// TwinCAT 3 PLC project SPS_Program
// ProgramVersion: 3.1.4023.0
// libraries:
//   Tc2_EtherCAT, * (Beckhoff Automation GmbH)
//   Tc2_Standard, * (Beckhoff Automation GmbH)
//   Tc2_System, * (Beckhoff Automation GmbH)
//   Tc3_Module, * (Beckhoff Automation GmbH)
// project tree:
//   DUTs/ eStates.TcDUT
//   / PlcTask.TcTTO
//   POUs/ FB_EcMasterState.TcPOU, FB_IOs.TcPOU, FB_LightControl.TcPOU, FB_LogicSupply.TcPOU, FB_PowerSupply.TcPOU, FB_SlaveName.TcPOU, FB_Start.TcPOU, FB_WatchPhotoelectricBarrier.TcPOU, FB_YesNo.TcPOU, MAIN.TcPOU
// real-time tasks:
//   TASK PlcTask: cycle T#10ms, priority 20, ADS port 350
// I/O:
//   DEVICE Gerät 1 (Beckhoff CCAT)
//   DEVICE Gerät 2 (EtherCAT), AmsNetId 10.200.20.140.3.1
//     Klemme 1 (EK1200) [EK1200-5000 EtherCAT Netzteil (2A E-Bus)]
//       Klemme 2 (EL1018) [EL1018 8K. Dig. Eingang 24V, 10µs]
//       Klemme 3 (EL1018) [EL1018 8K. Dig. Eingang 24V, 10µs]
//       Klemme 4 (EL1018) [EL1018 8K. Dig. Eingang 24V, 10µs]
//       Klemme 5 (EL1018) [EL1018 8K. Dig. Eingang 24V, 10µs]
//       Klemme 6 (EL4104) [EL4104 4Ch. Ana. Ausgang 0-10V, 16bit]
//       Klemme 7 (EL3064) [EL3064 4Ch. Ana. Input 0-10V]
//       Klemme 8 (EL2068) [EL2068 8Ch. Dig Output 24V, 0.5A]
//       Klemme 9 (EL2068) [EL2068 8Ch. Dig Output 24V, 0.5A]
//       Klemme 10 (EL2068) [EL2068 8Ch. Dig Output 24V, 0.5A]
//       Klemme 11 (EL2068) [EL2068 8Ch. Dig Output 24V, 0.5A]
//       Klemme 12 (EL9011) [EL9011 Endklemme]
//   DEVICE Gerät 3 (EtherCAT), AmsNetId 10.200.20.140.4.1
//     Antrieb 14 (SOMANET Node) [SOMANET Node CiA402 Antrieb]
//       modules: Module 1 (CiA402 Dictionary)
//     Antrieb 15 (SOMANET Node) [SOMANET Node CiA402 Antrieb]
//       modules: Module 1 (CiA402 Dictionary)
// variable links:
//   SPS_Program/SPS_Program Instance <-> Device 2 (EtherCAT)/Term 1 (EK1200)/Term 10 (EL2068)
//     PlcTask Outputs/MAIN.bA83_1 <-> DOS RxPDO-Map Outputs Ch.01/Output
//     PlcTask Outputs/MAIN.bA83_2 <-> DOS RxPDO-Map Outputs Ch.03/Output
//     PlcTask Outputs/MAIN.bA83_3 <-> DOS RxPDO-Map Outputs Ch.05/Output
//     PlcTask Outputs/MAIN.bA83_4 <-> DOS RxPDO-Map Outputs Ch.07/Output
//     PlcTask Outputs/MAIN.bA83_5 <-> DOS RxPDO-Map Outputs Ch.02/Output
//     PlcTask Outputs/MAIN.bA83_6 <-> DOS RxPDO-Map Outputs Ch.04/Output
//     PlcTask Outputs/MAIN.bA83_7 <-> DOS RxPDO-Map Outputs Ch.06/Output
//     PlcTask Outputs/MAIN.bA83_8 <-> DOS RxPDO-Map Outputs Ch.08/Output
//   SPS_Program/SPS_Program Instance <-> Device 2 (EtherCAT)/Term 1 (EK1200)/Term 11 (EL2068)
//     PlcTask Outputs/MAIN.bA84_1 <-> DOS RxPDO-Map Outputs Ch.01/Output
//     PlcTask Outputs/MAIN.bA84_2 <-> DOS RxPDO-Map Outputs Ch.02/Output
//     PlcTask Outputs/MAIN.bA84_3 <-> DOS RxPDO-Map Outputs Ch.03/Output
//     PlcTask Outputs/MAIN.bA84_4 <-> DOS RxPDO-Map Outputs Ch.04/Output
//     PlcTask Outputs/MAIN.bA84_5 <-> DOS RxPDO-Map Outputs Ch.05/Output
//     PlcTask Outputs/MAIN.bA84_6 <-> DOS RxPDO-Map Outputs Ch.06/Output
//     PlcTask Outputs/MAIN.bA84_8 <-> DOS RxPDO-Map Outputs Ch.08/Output
//     PlcTask Outputs/MAIN.bA85_7 <-> DOS RxPDO-Map Outputs Ch.07/Output
//   SPS_Program/SPS_Program Instance <-> Device 2 (EtherCAT)/Term 1 (EK1200)/Term 2 (EL1018)
//     PlcTask Inputs/MAIN.bA61_1 <-> Channel 1/Input
//     PlcTask Inputs/MAIN.bA61_2 <-> Channel 3/Input
//     PlcTask Inputs/MAIN.bA61_3 <-> Channel 5/Input
//     PlcTask Inputs/MAIN.bA61_4 <-> Channel 7/Input
//     PlcTask Inputs/MAIN.bA61_5 <-> Channel 2/Input
//     PlcTask Inputs/MAIN.bA61_6 <-> Channel 4/Input
//     PlcTask Inputs/MAIN.bA61_7 <-> Channel 6/Input
//     PlcTask Inputs/MAIN.bA61_8 <-> Channel 8/Input
//   SPS_Program/SPS_Program Instance <-> Device 2 (EtherCAT)/Term 1 (EK1200)/Term 3 (EL1018)
//     PlcTask Inputs/MAIN.bA62_1 <-> Channel 1/Input
//   SPS_Program/SPS_Program Instance <-> Device 2 (EtherCAT)/Term 1 (EK1200)/Term 4 (EL1018)
//     PlcTask Inputs/MAIN.bA63_1 <-> Channel 1/Input
//   SPS_Program/SPS_Program Instance <-> Device 2 (EtherCAT)/Term 1 (EK1200)/Term 5 (EL1018)
//     PlcTask Inputs/MAIN.bA64_1 <-> Channel 1/Input
//     PlcTask Inputs/MAIN.bA64_2 <-> Channel 3/Input
//     PlcTask Inputs/MAIN.bA64_3 <-> Channel 5/Input
//     PlcTask Inputs/MAIN.bA64_4 <-> Channel 7/Input
//     PlcTask Inputs/MAIN.bA64_5 <-> Channel 2/Input
//     PlcTask Inputs/MAIN.bA64_6 <-> Channel 4/Input
//     PlcTask Inputs/MAIN.bA64_7 <-> Channel 6/Input
//     PlcTask Inputs/MAIN.bA64_8 <-> Channel 8/Input
//   SPS_Program/SPS_Program Instance <-> Device 2 (EtherCAT)/Term 1 (EK1200)/Term 6 (EL4104)
//     PlcTask Outputs/MAIN.nA71_1 <-> AO Output Channel 1/Analog output
//     PlcTask Outputs/MAIN.nA71_3 <-> AO Output Channel 3/Analog output
//     PlcTask Outputs/MAIN.nA71_5 <-> AO Output Channel 2/Analog output
//     PlcTask Outputs/MAIN.nA71_7 <-> AO Output Channel 4/Analog output
//   SPS_Program/SPS_Program Instance <-> Device 2 (EtherCAT)/Term 1 (EK1200)/Term 7 (EL3064)
//     PlcTask Inputs/MAIN.nA72_1 <-> AI Standard Channel 1/Value
//     PlcTask Inputs/MAIN.nA72_3 <-> AI Standard Channel 3/Value
//     PlcTask Inputs/MAIN.nA72_5 <-> AI Standard Channel 2/Value
//     PlcTask Inputs/MAIN.nA72_7 <-> AI Standard Channel 4/Value
//   SPS_Program/SPS_Program Instance <-> Device 2 (EtherCAT)/Term 1 (EK1200)/Term 8 (EL2068)
//     PlcTask Outputs/MAIN.bA81_1 <-> DOS RxPDO-Map Outputs Ch.01/Output
//     PlcTask Outputs/MAIN.bA81_2 <-> DOS RxPDO-Map Outputs Ch.03/Output
//     PlcTask Outputs/MAIN.bA81_3 <-> DOS RxPDO-Map Outputs Ch.05/Output
//     PlcTask Outputs/MAIN.bA81_4 <-> DOS RxPDO-Map Outputs Ch.07/Output
//     PlcTask Outputs/MAIN.bA81_5 <-> DOS RxPDO-Map Outputs Ch.02/Output
//     PlcTask Outputs/MAIN.bA81_6 <-> DOS RxPDO-Map Outputs Ch.04/Output
//     PlcTask Outputs/MAIN.bA81_7 <-> DOS RxPDO-Map Outputs Ch.06/Output
//     PlcTask Outputs/MAIN.bA81_8 <-> DOS RxPDO-Map Outputs Ch.08/Output
//   SPS_Program/SPS_Program Instance <-> Device 2 (EtherCAT)/Term 1 (EK1200)/Term 9 (EL2068)
//     PlcTask Outputs/MAIN.bA82_1 <-> DOS RxPDO-Map Outputs Ch.01/Output
//     PlcTask Outputs/MAIN.bA82_2 <-> DOS RxPDO-Map Outputs Ch.03/Output
//     PlcTask Outputs/MAIN.bA82_3 <-> DOS RxPDO-Map Outputs Ch.05/Output
//     PlcTask Outputs/MAIN.bA82_4 <-> DOS RxPDO-Map Outputs Ch.07/Output
//     PlcTask Outputs/MAIN.bA82_5 <-> DOS RxPDO-Map Outputs Ch.02/Output
//     PlcTask Outputs/MAIN.bA82_6 <-> DOS RxPDO-Map Outputs Ch.04/Output
//     PlcTask Outputs/MAIN.bA82_7 <-> DOS RxPDO-Map Outputs Ch.06/Output
//     PlcTask Outputs/MAIN.bA82_8 <-> DOS RxPDO-Map Outputs Ch.08/Output
//   SPS_Program/SPS_Program Instance <-> Device 3 (EtherCAT)/Drive 14 (SOMANET Node)
//     PlcTask Inputs/MAIN.statusword_node_13 <-> TxPDO Mapping 1/Statusword
//   SPS_Program/SPS_Program Instance <-> Device 3 (EtherCAT)/Drive 15 (SOMANET Node)
//     PlcTask Inputs/MAIN.statusword_node_14 <-> TxPDO Mapping 1/Statusword

CONFIGURATION SPS_Program
    RESOURCE PLC ON TwinCAT3
        TASK PlcTask(INTERVAL := T#10ms, PRIORITY := 20);
        PROGRAM MAIN WITH PlcTask : MAIN;
    END_RESOURCE
END_CONFIGURATION

// ---- DUTs/eStates.TcDUT
{attribute 'qualified_only'}
{attribute 'strict'}
TYPE eStates :
(
	INIT,
	START_EXECUTION,
	EXECUTING,
	DONE
);
END_TYPE

// ---- POUs/MAIN.TcPOU
PROGRAM MAIN
//A61
VAR
	{attribute 'TcLinkTo' := 'TIID^Device 2 (EtherCAT)^Term 1 (EK1200)^Term 2 (EL1018)^Channel 1^Input'} 
	bA61_1		AT %I* 				: BOOL;
	{attribute 'TcLinkTo' := 'TIID^Device 2 (EtherCAT)^Term 1 (EK1200)^Term 2 (EL1018)^Channel 3^Input'} 
	bA61_2		AT %I* 				: BOOL;
	{attribute 'TcLinkTo' := 'TIID^Device 2 (EtherCAT)^Term 1 (EK1200)^Term 2 (EL1018)^Channel 5^Input'} 
	bA61_3		AT %I* 				: BOOL; 
	{attribute 'TcLinkTo' := 'TIID^Device 2 (EtherCAT)^Term 1 (EK1200)^Term 2 (EL1018)^Channel 7^Input'} 	
	bA61_4		AT %I* 				: BOOL;	
	{attribute 'TcLinkTo' := 'TIID^Device 2 (EtherCAT)^Term 1 (EK1200)^Term 2 (EL1018)^Channel 2^Input'} 		
	bA61_5		AT %I* 				: BOOL;
	{attribute 'TcLinkTo' := 'TIID^Device 2 (EtherCAT)^Term 1 (EK1200)^Term 2 (EL1018)^Channel 4^Input'}	
	bA61_6		AT %I* 				: BOOL;
	{attribute 'TcLinkTo' := 'TIID^Device 2 (EtherCAT)^Term 1 (EK1200)^Term 2 (EL1018)^Channel 6^Input'}	
	bA61_7		AT %I* 				: BOOL;
	{attribute 'TcLinkTo' := 'TIID^Device 2 (EtherCAT)^Term 1 (EK1200)^Term 2 (EL1018)^Channel 8^Input'}
	bA61_8		AT %I* 				: BOOL;
	bSetEnable_SlaveName: BOOL;
END_VAR


//A62
VAR
	{attribute 'TcLinkTo' := 'TIID^Device 2 (EtherCAT)^Term 1 (EK1200)^Term 3 (EL1018)^Channel 1^Input'} 
	bA62_1		AT %I* 				: BOOL;
	{attribute 'TcLinkTo' := 'TIID^Device 3 (EtherCAT)^Term 1 (EK1200)^Term 3 (EL1018)^Channel 3^Input'} 
	bA62_2		AT %I* 				: BOOL;
	{attribute 'TcLinkTo' := 'TIID^Device 3 (EtherCAT)^Term 1 (EK1200)^Term 3 (EL1018)^Channel 5^Input'} 
	bA62_3		AT %I* 				: BOOL; 
	{attribute 'TcLinkTo' := 'TIID^Device 3 (EtherCAT)^Term 1 (EK1200)^Term 3 (EL1018)^Channel 7^Input'} 	
	bA62_4		AT %I* 				: BOOL;	
	{attribute 'TcLinkTo' := 'TIID^Device 3 (EtherCAT)^Term 1 (EK1200)^Term 3 (EL1018)^Channel 2^Input'} 		
	bA62_5		AT %I* 				: BOOL;
	{attribute 'TcLinkTo' := 'TIID^Device 3 (EtherCAT)^Term 1 (EK1200)^Term 3 (EL1018)^Channel 4^Input'}	
	bA62_6		AT %I* 				: BOOL;
	{attribute 'TcLinkTo' := 'TIID^Device 3 (EtherCAT)^Term 1 (EK1200)^Term 3 (EL1018)^Channel 6^Input'}	
	bA62_7		AT %I* 				: BOOL;
	{attribute 'TcLinkTo' := 'TIID^Device 3 (EtherCAT)^Term 1 (EK1200)^Term 3 (EL1018)^Channel 8^Input'}
	bA62_8		AT %I* 				: BOOL;
END_VAR


//A63
VAR
	{attribute 'TcLinkTo' := 'TIID^Device 2 (EtherCAT)^Term 1 (EK1200)^Term 4 (EL1018)^Channel 1^Input'} 
	bA63_1		AT %I* 				: BOOL;
	{attribute 'TcLinkTo' := 'TIID^Device 3 (EtherCAT)^Term 1 (EK1200)^Term 4 (EL1018)^Channel 3^Input'} 
	bA63_2		AT %I* 				: BOOL;
	{attribute 'TcLinkTo' := 'TIID^Device 3 (EtherCAT)^Term 1 (EK1200)^Term 4 (EL1018)^Channel 5^Input'} 
	bA63_3		AT %I* 				: BOOL; 
	{attribute 'TcLinkTo' := 'TIID^Device 3 (EtherCAT)^Term 1 (EK1200)^Term 4 (EL1018)^Channel 7^Input'} 	
	bA63_4		AT %I* 				: BOOL;	
	{attribute 'TcLinkTo' := 'TIID^Device 3 (EtherCAT)^Term 1 (EK1200)^Term 4 (EL1018)^Channel 2^Input'} 		
	bA63_5		AT %I* 				: BOOL;
	{attribute 'TcLinkTo' := 'TIID^Device 3 (EtherCAT)^Term 1 (EK1200)^Term 4 (EL1018)^Channel 4^Input'}	
	bA63_6		AT %I* 				: BOOL;
	{attribute 'TcLinkTo' := 'TIID^Device 3 (EtherCAT)^Term 1 (EK1200)^Term 4 (EL1018)^Channel 6^Input'}	
	bA63_7		AT %I* 				: BOOL;
	{attribute 'TcLinkTo' := 'TIID^Device 3 (EtherCAT)^Term 1 (EK1200)^Term 4 (EL1018)^Channel 8^Input'}
	bA63_8		AT %I* 				: BOOL;
END_VAR


//A64
VAR
	{attribute 'TcLinkTo' := 'TIID^Device 2 (EtherCAT)^Term 1 (EK1200)^Term 5 (EL1018)^Channel 1^Input'}
	bA64_1		AT %I*				: BOOL; 
	{attribute 'TcLinkTo' := 'TIID^Device 2 (EtherCAT)^Term 1 (EK1200)^Term 5 (EL1018)^Channel 3^Input'}	
	bA64_2		AT %I* 				: BOOL;	
	{attribute 'TcLinkTo' := 'TIID^Device 2 (EtherCAT)^Term 1 (EK1200)^Term 5 (EL1018)^Channel 5^Input'}
	bA64_3		AT %I* 				: BOOL;
	{attribute 'TcLinkTo' := 'TIID^Device 2 (EtherCAT)^Term 1 (EK1200)^Term 5 (EL1018)^Channel 7^Input'}
	bA64_4		AT %I* 				: BOOL;
	{attribute 'TcLinkTo' := 'TIID^Device 2 (EtherCAT)^Term 1 (EK1200)^Term 5 (EL1018)^Channel 2^Input'}
	bA64_5		AT %I* 				: BOOL;
	{attribute 'TcLinkTo' := 'TIID^Device 2 (EtherCAT)^Term 1 (EK1200)^Term 5 (EL1018)^Channel 4^Input'}
	bA64_6		AT %I* 				: BOOL;
	{attribute 'TcLinkTo' := 'TIID^Device 2 (EtherCAT)^Term 1 (EK1200)^Term 5 (EL1018)^Channel 6^Input'}	
	bA64_7		AT %I* 				: BOOL;
	{attribute 'TcLinkTo' := 'TIID^Device 2 (EtherCAT)^Term 1 (EK1200)^Term 5 (EL1018)^Channel 8^Input'}
	bA64_8		AT %I* 				: BOOL;	
END_VAR


//A71
VAR	
	{attribute 'TcLinkTo' := 'TIID^Device 2 (EtherCAT)^Term 1 (EK1200)^Term 6 (EL4104)^AO Output Channel 1^Analog output'} 
	nA71_1		AT %Q* 				: UINT;
	{attribute 'TcLinkTo' := 'TIID^Device 2 (EtherCAT)^Term 1 (EK1200)^Term 6 (EL4104)^AO Output Channel 3^Analog output'} 
	nA71_3		AT %Q* 				: UINT;	
	{attribute 'TcLinkTo' := 'TIID^Device 2 (EtherCAT)^Term 1 (EK1200)^Term 6 (EL4104)^AO Output Channel 2^Analog output'} 
	nA71_5		AT %Q* 				: UINT;	
	{attribute 'TcLinkTo' := 'TIID^Device 2 (EtherCAT)^Term 1 (EK1200)^Term 6 (EL4104)^AO Output Channel 4^Analog output'} 
	nA71_7		AT %Q* 				: UINT;		
END_VAR


//A72
VAR
	{attribute 'TcLinkTo' := 'TIID^Device 2 (EtherCAT)^Term 1 (EK1200)^Term 7 (EL3064)^AI Standard Channel 1^Value'}
	nA72_1		AT %I* 				: UINT;	
	{attribute 'TcLinkTo' := 'TIID^Device 2 (EtherCAT)^Term 1 (EK1200)^Term 7 (EL3064)^AI Standard Channel 3^Value'}
 	nA72_3		AT %I* 				: UINT;	
	{attribute 'TcLinkTo' := 'TIID^Device 2 (EtherCAT)^Term 1 (EK1200)^Term 7 (EL3064)^AI Standard Channel 2^Value'}
	nA72_5		AT %I* 				: UINT;
	{attribute 'TcLinkTo' := 'TIID^Device 2 (EtherCAT)^Term 1 (EK1200)^Term 7 (EL3064)^AI Standard Channel 4^Value'}	
	nA72_7		AT %I* 				: UINT;	
END_VAR


//A81
VAR
	{attribute 'TcLinkTo' := 'TIID^Device 2 (EtherCAT)^Term 1 (EK1200)^Term 8 (EL2068)^DOS RxPDO-Map Outputs Ch.01^Output'}	
	bA81_1		AT %Q* 				: BOOL;
	{attribute 'TcLinkTo' := 'TIID^Device 2 (EtherCAT)^Term 1 (EK1200)^Term 8 (EL2068)^DOS RxPDO-Map Outputs Ch.03^Output'}		
	bA81_2		AT %Q* 				: BOOL;
	{attribute 'TcLinkTo' := 'TIID^Device 2 (EtherCAT)^Term 1 (EK1200)^Term 8 (EL2068)^DOS RxPDO-Map Outputs Ch.05^Output'}		
	bA81_3		AT %Q* 				: BOOL;
	{attribute 'TcLinkTo' := 'TIID^Device 2 (EtherCAT)^Term 1 (EK1200)^Term 8 (EL2068)^DOS RxPDO-Map Outputs Ch.07^Output'} 
	bA81_4		AT %Q* 				: BOOL; 
	{attribute 'TcLinkTo' := 'TIID^Device 2 (EtherCAT)^Term 1 (EK1200)^Term 8 (EL2068)^DOS RxPDO-Map Outputs Ch.02^Output'}
	bA81_5		AT %Q* 				: BOOL; 
	{attribute 'TcLinkTo' := 'TIID^Device 2 (EtherCAT)^Term 1 (EK1200)^Term 8 (EL2068)^DOS RxPDO-Map Outputs Ch.04^Output'}
	bA81_6		AT %Q* 				: BOOL;	
	{attribute 'TcLinkTo' := 'TIID^Device 2 (EtherCAT)^Term 1 (EK1200)^Term 8 (EL2068)^DOS RxPDO-Map Outputs Ch.06^Output'}
	bA81_7		AT %Q* 				: BOOL; 
	{attribute 'TcLinkTo' := 'TIID^Device 2 (EtherCAT)^Term 1 (EK1200)^Term 8 (EL2068)^DOS RxPDO-Map Outputs Ch.08^Output'}
	bA81_8		AT %Q* 				: BOOL; 
END_VAR


//A82
VAR
	{attribute 'TcLinkTo' := 'TIID^Device 2 (EtherCAT)^Term 1 (EK1200)^Term 9 (EL2068)^DOS RxPDO-Map Outputs Ch.01^Output'}
	bA82_1		AT %Q* 				: BOOL;
	{attribute 'TcLinkTo' := 'TIID^Device 2 (EtherCAT)^Term 1 (EK1200)^Term 9 (EL2068)^DOS RxPDO-Map Outputs Ch.03^Output'}
	bA82_2		AT %Q* 				: BOOL;
	{attribute 'TcLinkTo' := 'TIID^Device 2 (EtherCAT)^Term 1 (EK1200)^Term 9 (EL2068)^DOS RxPDO-Map Outputs Ch.05^Output'}
	bA82_3		AT %Q* 				: BOOL;
	{attribute 'TcLinkTo' := 'TIID^Device 2 (EtherCAT)^Term 1 (EK1200)^Term 9 (EL2068)^DOS RxPDO-Map Outputs Ch.07^Output'}
	bA82_4		AT %Q* 				: BOOL;
	{attribute 'TcLinkTo' := 'TIID^Device 2 (EtherCAT)^Term 1 (EK1200)^Term 9 (EL2068)^DOS RxPDO-Map Outputs Ch.02^Output'}
	bA82_5		AT %Q* 				: BOOL;
	{attribute 'TcLinkTo' := 'TIID^Device 2 (EtherCAT)^Term 1 (EK1200)^Term 9 (EL2068)^DOS RxPDO-Map Outputs Ch.04^Output'}
	bA82_6		AT %Q* 				: BOOL;
	{attribute 'TcLinkTo' := 'TIID^Device 2 (EtherCAT)^Term 1 (EK1200)^Term 9 (EL2068)^DOS RxPDO-Map Outputs Ch.06^Output'}
	bA82_7		AT %Q* 				: BOOL;
	{attribute 'TcLinkTo' := 'TIID^Device 2 (EtherCAT)^Term 1 (EK1200)^Term 9 (EL2068)^DOS RxPDO-Map Outputs Ch.08^Output'}
	bA82_8		AT %Q* 				: BOOL;
END_VAR


//A83
VAR
	{attribute 'TcLinkTo' := 'TIID^Device 2 (EtherCAT)^Term 1 (EK1200)^Term 10 (EL2068)^DOS RxPDO-Map Outputs Ch.01^Output'}
	bA83_1		AT %Q* 				: BOOL;
	{attribute 'TcLinkTo' := 'TIID^Device 2 (EtherCAT)^Term 1 (EK1200)^Term 10 (EL2068)^DOS RxPDO-Map Outputs Ch.03^Output'}
	bA83_2		AT %Q* 				: BOOL;
	{attribute 'TcLinkTo' := 'TIID^Device 2 (EtherCAT)^Term 1 (EK1200)^Term 10 (EL2068)^DOS RxPDO-Map Outputs Ch.05^Output'}
	bA83_3		AT %Q* 				: BOOL;
	{attribute 'TcLinkTo' := 'TIID^Device 2 (EtherCAT)^Term 1 (EK1200)^Term 10 (EL2068)^DOS RxPDO-Map Outputs Ch.07^Output'}
	bA83_4		AT %Q* 				: BOOL;
	{attribute 'TcLinkTo' := 'TIID^Device 2 (EtherCAT)^Term 1 (EK1200)^Term 10 (EL2068)^DOS RxPDO-Map Outputs Ch.02^Output'}
	bA83_5		AT %Q* 				: BOOL;
	{attribute 'TcLinkTo' := 'TIID^Device 2 (EtherCAT)^Term 1 (EK1200)^Term 10 (EL2068)^DOS RxPDO-Map Outputs Ch.04^Output'}
	bA83_6		AT %Q* 				: BOOL;
	{attribute 'TcLinkTo' := 'TIID^Device 2 (EtherCAT)^Term 1 (EK1200)^Term 10 (EL2068)^DOS RxPDO-Map Outputs Ch.06^Output'}
	bA83_7		AT %Q* 				: BOOL;
	{attribute 'TcLinkTo' := 'TIID^Device 2 (EtherCAT)^Term 1 (EK1200)^Term 10 (EL2068)^DOS RxPDO-Map Outputs Ch.08^Output'}
	bA83_8		AT %Q* 				: BOOL;	
END_VAR


//A84
//TODO
VAR	
	{attribute 'TcLinkTo' := 'TIID^Device 2 (EtherCAT)^Term 1 (EK1200)^Term 11 (EL2068)^DOS RxPDO-Map Outputs Ch.01^Output'}
	bA84_1		AT %Q* 				: BOOL;
	{attribute 'TcLinkTo' := 'TIID^Device 2 (EtherCAT)^Term 1 (EK1200)^Term 11 (EL2068)^DOS RxPDO-Map Outputs Ch.02^Output'}
	bA84_2		AT %Q* 				: BOOL;
	{attribute 'TcLinkTo' := 'TIID^Device 2 (EtherCAT)^Term 1 (EK1200)^Term 11 (EL2068)^DOS RxPDO-Map Outputs Ch.03^Output'}
	bA84_3		AT %Q* 				: BOOL;	
	{attribute 'TcLinkTo' := 'TIID^Device 2 (EtherCAT)^Term 1 (EK1200)^Term 11 (EL2068)^DOS RxPDO-Map Outputs Ch.04^Output'}
	bA84_4		AT %Q* 				: BOOL;
	{attribute 'TcLinkTo' := 'TIID^Device 2 (EtherCAT)^Term 1 (EK1200)^Term 11 (EL2068)^DOS RxPDO-Map Outputs Ch.05^Output'}
	bA84_5		AT %Q* 				: BOOL;
	{attribute 'TcLinkTo' := 'TIID^Device 2 (EtherCAT)^Term 1 (EK1200)^Term 11 (EL2068)^DOS RxPDO-Map Outputs Ch.06^Output'}
	bA84_6		AT %Q* 				: BOOL;
	{attribute 'TcLinkTo' := 'TIID^Device 2 (EtherCAT)^Term 1 (EK1200)^Term 11 (EL2068)^DOS RxPDO-Map Outputs Ch.07^Output'}
	bA85_7		AT %Q* 				: BOOL;
	{attribute 'TcLinkTo' := 'TIID^Device 2 (EtherCAT)^Term 1 (EK1200)^Term 11 (EL2068)^DOS RxPDO-Map Outputs Ch.08^Output'}
	bA84_8		AT %Q* 				: BOOL;
END_VAR

VAR
	fbLightControlLeft				: FB_LightControl;
	fbLightControlRight				: FB_LightControl;
	fbPowerSupplyLeft				: FB_PowerSupply;
	fbStartLeft						: FB_Start;
	fbLogicSupplyLeft				: FB_LogicSupply;
	fbLogicSupplyRight				: FB_LogicSupply;
	fbYesNoLeft						: FB_YesNo;
	fbYesNoRight					: FB_YesNo;
	fbIOsLeft						: FB_IOs;
	fbIOsRight						: FB_IOs;
	fbWatchPhotoelectricBarrierLeft	: FB_WatchPhotoelectricBarrier;
	fbSTOLeft						: FB_LogicSupply;
	
	fbOblacBoxLeft					: FB_LogicSupply;
	fbOblacBoxRight					: FB_LogicSupply;
	
	fbReferenceControlerLeft		: FB_LogicSupply;
	fbReferenceControlerRight		: FB_LogicSupply;
	
	fbEcMasterStateLeft : FB_EcMasterState(sNetId := '5.124.224.126.4.1');
	//fbEcMasterStateRight : FB_EcMasterState(sNetId := '5.124.224.126.6.1');
	
	fbSlaveNameLeft : FB_SlaveName(sNetId := '5.124.224.126.4.1');
	//fbSlaveNameRight : FB_SlaveName(sNetId := '5.124.224.126.6.1');
END_VAR

VAR
	nTargetCurrentLeft				: UDINT;
	nTargetVoltageLeft				: UDINT;
	nTargetPowerLeft				: UDINT;
	nCurrentLeft					: UDINT;
	nVoltageLeft					: UDINT;
END_VAR

VAR
	bTestGreen						: BOOL;
	bTestRed						: BOOL;
	bTestWhite						: BOOL;
	bTestYellow						: BOOL;
	bSwitchOff						: BOOL;
	bTestLogicOn					: BOOL;
	bTestLogicOff					: BOOL;
	bTestPowerSupply				: BOOL;
	bReset							: BOOL;
	bSetPowVolCurr					: BOOL;
	bSwitchOnPowerSupply			: BOOL;
	bSwitchOffPowerSupply			: BOOL;
	
	bReadName : BOOL := FALSE;
	
	bGotAnswer : BOOL := FALSE;
	
	{attribute 'TcLinkTo' := 'TIID^Device 3 (EtherCAT)^Drive 14 (SOMANET Node)^TxPDO Mapping 1^Statusword'}
	statusword_node_13 AT %I* : UINT;
	
	{attribute 'TcLinkTo' := 'TIID^Device 3 (EtherCAT)^Drive 15 (SOMANET Node)^TxPDO Mapping 1^Statusword'}
	statusword_node_14 AT %I* : UINT;
	
	bInit : BOOL := FALSE; //for switching master into init
	
	bSetEnable : BOOL := FALSE;
	
END_VAR

fbOblacBoxLeft(bSwitchOn := bA83_1);
fbReferenceControlerLeft(bSwitchOn := bA83_2);
	
fbOblacBoxRight(bSwitchOn := bA83_3);
fbReferenceControlerRight(bSwitchOn := bA83_4);

///////////////////Logic-Supply/////////////////////////////
fbLogicSupplyLeft(bSwitchOn := bA82_3);		
fbLogicSupplyRight (bSwitchOn := bA82_7);

IF NOT bInit THEN
	fbOblacBoxLeft.SwitchOn();
	fbReferenceControlerLeft.SwitchOff();
	fbEcMasterStateLeft.DisableMaster();
	bInit := TRUE;
END_IF

//////////////////////EC-IN-OUT/////////////////////////////////
fbSlaveNameLeft();
//fbSlaveNameRight();
fbEcMasterStateLeft();
//fbEcMasterStateRight();
					
/////////////////////Power-Supply///////////////////////////////

IF bSwitchOnPowerSupply THEN
	fbPowerSupplyLeft.SwitchOn();
	bSwitchOnPowerSupply := FALSE;
END_IF

IF bSwitchOffPowerSupply THEN
	fbPowerSupplyLeft.SwitchOff();
	bSwitchOffPowerSupply := FALSE;
END_IF


fbPowerSupplyLeft.TargetCurrent := nTargetCurrentLeft;
fbPowerSupplyLeft.TargetVoltage := nTargetVoltageLeft;
fbPowerSupplyLeft.TargetPower := nTargetPowerLeft;
bSetPowVolCurr := FALSE;

fbPowerSupplyLeft(nMaxVoltage := 80000,
					nMaxPower := 150000,
					nMaxCurrent := 50000,
					nCurrentFromPowerSupply := nA72_3,
					nVoltageFromPowerSupply := nA72_5,
					nReferenceVoltage := nA72_1,
					bREMSB => bA81_5,
					nVoltage => nA71_1,
					nCurrent => nA71_5,
					nPower => nA71_3);
					
nCurrentLeft := fbPowerSupplyLeft.CurrentCurrent;
nVoltageLeft := fbPowerSupplyLeft.CurrentVoltage;



///////////////////STO-Supply/////////////////////////////
fbSTOLeft(bSwitchOn := bA82_5);


/////////////////////Light-Control///////////////////////////////
fbLightControlLeft (bTrig1 := bA84_1,  //weiß
					bTrig2 := bA84_3,	//Grau
				 	bTrig3 := bA84_2);	//Schwarz
				 
fbLightControlRight(bTrig1	:= bA84_4,	//weiß
					bTrig2	:= bA84_6,	//grau
					bTrig3	:= bA84_5);	//schwarz
					
/////////////////////Physical-Buttons///////////////////////////
fbStartLeft(bSwitchOn := bA64_1,
			bSwitchOff := bA64_2);
			
fbYesNoLeft(bYes := bA64_1,
			bNo := bA64_2,
			bGotAnswer => bGotAnswer);
			
IF bReset THEN
	fbYesNoLeft.Reset();
	bReset := FALSE;
END_IF
			
/////////////////////Photoelectric-Barrier///////////////////////
fbWatchPhotoelectricBarrierLeft(nInterrupted := nA72_7);

//IF fbWatchPhotoelectricBarrierLeft.bInterrupted THEN
//	fbPowerSupplyLeft.SwitchOff();
//	fbLogicSupplyLeft.SwitchOff();
//END_IF


///////////////////////////Testing//////////////////////////////////

IF bSetEnable THEN
	fbEcMasterStateLeft.EnableMaster();
	bSetEnable := FALSE;
END_IF

IF bSetEnable_SlaveName THEN
	fbSlaveNameLeft.CheckName('Testmotor');
	bSetEnable_SlaveName := FALSE;
END_IF

END_PROGRAM

// ---- POUs/FB_LightControl.TcPOU
FUNCTION_BLOCK FB_LightControl
VAR_IN_OUT
	bTrig1		:	BOOL;
	bTrig2		: 	BOOL;
	bTrig3		: 	BOOL;
END_VAR

{attribute 'TcRpcEnable'}
METHOD Green
bTrig1	:= FALSE;
bTrig2	:= TRUE;
bTrig3	:= FALSE;
END_METHOD

{attribute 'TcRpcEnable'}
METHOD Red
bTrig1	:= TRUE;
bTrig2	:= FALSE;
bTrig3	:= FALSE;
END_METHOD

{attribute 'TcRpcEnable'}
METHOD SwitchOff : BOOL
bTrig1	:= FALSE;
bTrig2	:= FALSE;
bTrig3	:= FALSE;
END_METHOD

{attribute 'TcRpcEnable'}
METHOD White : BOOL
bTrig1	:= FALSE;
bTrig2	:= FALSE;
bTrig3	:= TRUE;
END_METHOD

{attribute 'TcRpcEnable'}
METHOD Yellow : BOOL
bTrig1	:= TRUE;
bTrig2	:= TRUE;
bTrig3	:= FALSE;
END_METHOD

END_FUNCTION_BLOCK

// ---- POUs/FB_PowerSupply.TcPOU
FUNCTION_BLOCK FB_PowerSupply
VAR_INPUT
	nMaxVoltage						: UDINT;
	nMaxPower						: DINT;
	nMaxCurrent						: UINT;
	
	nCurrentFromPowerSupply			: UINT;
	nVoltageFromPowerSupply			: UINT;
	
	nReferenceVoltage				: UINT;  //Reference Voltage 
END_VAR

VAR_OUTPUT
	nVoltage						: UINT;
	nCurrent						: UINT;
	nPower							: UINT;
	bREMSB							: BOOL;
END_VAR
VAR
	nTargetVoltage					: UDINT;
	nTargetPower					: UDINT;
	nTargetCurrent					: UDINT;
END_VAR

bREMSB := TRUE;

PROPERTY CurrentCurrent : UINT
GET
IF nReferenceVoltage = 0 THEN
	CurrentCurrent := 0;
ELSE
	CurrentCurrent := nCurrentFromPowerSupply * nMaxCurrent/nReferenceVoltage;
END_IF
END_GET
END_PROPERTY

PROPERTY CurrentVoltage : UINT
GET
IF nReferenceVoltage = 0 THEN
	CurrentVoltage := 0;
ELSE
	CurrentVoltage := UDINT_TO_UINT(nVoltageFromPowerSupply * nMaxVoltage/nReferenceVoltage);
END_IF
END_GET
END_PROPERTY

{attribute 'TcRpcEnable'}
METHOD SwitchOff
nVoltage := 0;
nCurrent := 0;
nPower := 0;
END_METHOD

{attribute 'TcRpcEnable'}
METHOD SwitchOn
nVoltage := UDINT_TO_UINT(nTargetVoltage);
nCurrent := UDINT_TO_UINT(nTargetCurrent);
nPower := UDINT_TO_UINT(nTargetPower);
END_METHOD

PROPERTY TargetCurrent : UDINT
GET
TargetCurrent := nTargetCurrent * nMaxCurrent/nReferenceVoltage;
END_GET
SET
IF TargetCurrent < nMaxCurrent THEN
	nTargetCurrent := TargetCurrent * nReferenceVoltage / nMaxCurrent;
ELSE
	nTargetCurrent := 32767;
END_IF
END_SET
END_PROPERTY

PROPERTY TargetPower : UDINT
GET
TargetPower := UDINT_TO_UINT(nTargetPower * nMaxPower/nReferenceVoltage);
END_GET
SET
IF TargetPower < nMaxPower THEN
	nTargetPower := UDINT_TO_UINT(TargetPower * nReferenceVoltage / nMaxPower);
ELSE
	nTargetPower := 32767;
END_IF
END_SET
END_PROPERTY

PROPERTY TargetVoltage : UDINT
GET
IF (nReferenceVoltage = 0) THEN
	TargetVoltage := 0;
ELSE
		TargetVoltage := nTargetVoltage * nMaxVoltage/nReferenceVoltage;
END_IF
END_GET
SET
IF TargetVoltage < nMaxVoltage THEN
	nTargetVoltage := TargetVoltage * nReferenceVoltage/nMaxVoltage;	
	//ADSLOGSTR(msgCtrlMask := ADSLOG_MSGTYPE_HINT, 
    //    	msgFmtStr   := 'Desired Voltage is lower than nMaxVoltage: %s', 
    //    	strArg      := UDINT_TO_STRING(TargetVoltage)
    //		);  
ELSE
	nTargetVoltage := 32767;
	//ADSLOGSTR(msgCtrlMask := ADSLOG_MSGTYPE_HINT, 
    //    	msgFmtStr   := 'Desired Voltage is higher than nMaxVoltage: %s', 
    //    	strArg      := UDINT_TO_STRING(TargetVoltage)
    //		);  
END_IF
END_SET
END_PROPERTY

END_FUNCTION_BLOCK

// ---- POUs/FB_Start.TcPOU
FUNCTION_BLOCK FB_Start
VAR_INPUT
	bSwitchOn				: BOOL;
	bSwitchOff				: BOOL;
END_VAR
VAR
	bSwitchedOn				: BOOL;
END_VAR

{attribute 'TcRpcEnable'}
METHOD SwitchOff
bSwitchedOn := FALSE;
END_METHOD

{attribute 'TcRpcEnable'}
METHOD SwitchOn : BOOL
VAR_INPUT
END_VAR
bSwitchedOn := TRUE;
END_METHOD

END_FUNCTION_BLOCK

// ---- POUs/FB_LogicSupply.TcPOU
FUNCTION_BLOCK FB_LogicSupply
VAR_IN_OUT
	bSwitchOn		: BOOL;
END_VAR

{attribute 'TcRpcEnable'}
METHOD SwitchOff
bSwitchOn := FALSE;
END_METHOD

{attribute 'TcRpcEnable'}
METHOD SwitchOn
bSwitchOn := TRUE;
END_METHOD

END_FUNCTION_BLOCK

// ---- POUs/FB_YesNo.TcPOU
FUNCTION_BLOCK FB_YesNo
VAR_INPUT
	bYes			: BOOL;
	bNo				: BOOL;
END_VAR
VAR_OUTPUT
	bAnswer			: BOOL;
	bGotAnswer		: BOOL;
END_VAR
VAR
	fTrig			: F_Trig;
	rTrig			: R_Trig;
END_VAR

rTrig(CLK := bYes);
fTrig(CLK := bNo);

IF (rTrig.Q OR fTrig.Q) THEN
	bGotAnswer := TRUE;
END_IF
IF bYes THEN
	bAnswer := TRUE;
END_IF

{attribute 'TcRpcEnable'}
METHOD Reset
bAnswer		:= FALSE;
bGotAnswer 	:= FALSE;
END_METHOD

END_FUNCTION_BLOCK

// ---- POUs/FB_IOs.TcPOU
FUNCTION_BLOCK FB_IOs
VAR_INPUT
END_VAR
VAR_OUTPUT
END_VAR
VAR
END_VAR

{attribute 'TcRpcEnable'}
METHOD Check : BOOL
VAR_INPUT
END_VAR
END_METHOD

END_FUNCTION_BLOCK

// ---- POUs/FB_WatchPhotoelectricBarrier.TcPOU
FUNCTION_BLOCK FB_WatchPhotoelectricBarrier
VAR_INPUT
	nInterrupted		: UINT;
END_VAR
VAR_OUTPUT
	bInterrupted		: BOOL;
END_VAR

IF nInterrupted < (32767 / 2) THEN
	bInterrupted := TRUE;
ELSE
	bInterrupted := FALSE;
END_IF

END_FUNCTION_BLOCK

// ---- POUs/FB_EcMasterState.TcPOU
FUNCTION_BLOCK FB_EcMasterState

VAR_INPUT
	sNetId           : T_AmsNetId; //:= '5.124.224.126.6.1';
END_VAR

VAR
    fbReqMasterState : FB_EcReqMasterState;
    bExecute         : BOOL;
	tTimeout		 : TIME := DEFAULT_ADS_TIMEOUT;
    ReqMasterState      : WORD;
	bBusy  			 : BOOL;
END_VAR

VAR_OUTPUT
    bError           : BOOL;
    nErrId           : UDINT;

	bStateChangeSuccessful : BOOL;//fertig bit
	bStateChangeOccurred : BOOL; //erfolgt bit
END_VAR

//other function blocks
VAR
	fTrig			: F_Trig;
END_VAR

VAR
	state : eStates := eStates.INIT;
END_VAR

// state machine

CASE state OF
    eStates.INIT: //default state
	
	        bStateChangeSuccessful := FALSE;
			
			bStateChangeOccurred := FALSE;
			bError := FALSE;
			nErrId := 0;
			//ADSLOGSTR(msgCtrlMask := ADSLOG_MSGTYPE_HINT, msgFmtStr   := 'occurred set false %s','');
			
        IF bExecute THEN

            bExecute := FALSE; // Verhindert erneutes Auslösen
            bStateChangeSuccessful := FALSE;
			
			bStateChangeOccurred := FALSE;
			
			fbReqMasterState(sNetId:= sNetId, bExecute:=FALSE, state:= ReqMasterState);
			
			state := eStates.START_EXECUTION;
        END_IF
        
    eStates.START_EXECUTION:
			fbReqMasterState(); //zustand abfragen
        IF NOT fbReqMasterState.bBusy THEN //nicht starten falls doch noch bussy
			fbReqMasterState(sNetId:= sNetId, bExecute:=TRUE, state:=ReqMasterState); //starten
			
            state := eStates.EXECUTING;

        END_IF

    eStates.EXECUTING:
	
		fbReqMasterState(); //Bussy flag update

		IF fbReqMasterState.bBusy THEN
			// Warten auf Abschluss der Operation
			// TODO hier timeout
		ELSE
            IF NOT fbReqMasterState.bError THEN
                bStateChangeSuccessful := TRUE;
											ADSLOGSTR(
        	msgCtrlMask := ADSLOG_MSGTYPE_HINT, 
        	msgFmtStr   := 'beendet ohne fehler %s','');
            ELSE
                bStateChangeSuccessful := FALSE;
				bError := fbReqMasterState.bError;
				nErrId := fbReqMasterState.nErrId;
							ADSLOGSTR(
        	msgCtrlMask := ADSLOG_MSGTYPE_HINT, 
        	msgFmtStr   := 'beendet mit fehler %s','');
            END_IF

			bStateChangeOccurred := TRUE; // Signalisieren, dass eine Änderung stattgefunden hat
            state := eStates.DONE;
        END_IF

    eStates.DONE:
	
	bExecute := FALSE;
    //waiting for reset ...  no automatic reset    
    //state := eStates.INIT;

ELSE
	state := eStates.INIT;
	
END_CASE;

{attribute 'TcRpcEnable'}
METHOD DisableMaster : BOOL
VAR_INPUT
END_VAR
//only works if state machine is in init mode
bExecute := TRUE;
ReqMasterState := EC_DEVICE_STATE_INIT;
END_METHOD

{attribute 'TcRpcEnable'}
METHOD EnableMaster : BOOL
VAR_INPUT
END_VAR

VAR
END_VAR
//only works if state machine is in init mode
bExecute := TRUE;
ReqMasterState := EC_DEVICE_STATE_OP;
END_METHOD

METHOD FB_init : BOOL
VAR_INPUT
    bInitRetains : BOOL; // if TRUE, the retain variables are initialized (warm start / cold start)
    bInCopyCode  : BOOL; // if TRUE, the instance afterwards gets moved into the copy code (online change)
	sNetId           : T_AmsNetId;
END_VAR
THIS^.sNetId := sNetId;
END_METHOD

{attribute 'TcRpcEnable'}
METHOD Reset : BOOL
VAR_INPUT
END_VAR
state := eStates.INIT;
END_METHOD

END_FUNCTION_BLOCK

// ---- POUs/FB_SlaveName.TcPOU
FUNCTION_BLOCK FB_SlaveName

VAR_INPUT
	sNetId     : T_AmsNetId;// := '5.124.224.126.6.1';	
END_VAR

VAR CONSTANT
	nSlaveAddr : UINT := 1002; //motor 2
    nIndex     : WORD := 16#20F2; //assigned name
    nSubIndex  : BYTE := 0;
END_VAR

VAR
	fbSdoRead  : FB_EcCoESdoRead;
    bExecute   : BOOL;

	
	state : eStates := eStates.INIT;
	RevSlaveName: STRING;
END_VAR

VAR_OUTPUT
	bError     : BOOL;
    nErrId     : UDINT;
	
	SlaveName : STRING;
	
	bReadSlaveNameOccurred : BOOL;
	bReadSlaveNameSuccessful : BOOL;
	bNameIsEqual : BOOL;
END_VAR

// state machine

CASE state OF
    eStates.INIT: //default state
	
	    bReadSlaveNameOccurred := FALSE;
        bReadSlaveNameSuccessful := FALSE;
		bNameIsEqual := FALSE;
		SlaveName := '';
		//RevSlaveName := '';
		
		
		fbSdoRead(sNetId:= sNetId,nSlaveAddr :=nSlaveAddr, nIndex:=nIndex,
				nSubIndex :=nSubIndex, pDstBuf:= ADR(SlaveName), cbBufLen:=SIZEOF(SlaveName), bExecute:=FALSE);
			
        IF bExecute THEN
            state := eStates.START_EXECUTION;
            bExecute := FALSE; // Verhindert erneutes Auslösen


			
			ADSLOGSTR(msgCtrlMask := ADSLOG_MSGTYPE_HINT, msgFmtStr   := 'executed %s','');
        END_IF
        
    eStates.START_EXECUTION:
	
		fbSdoRead();
	
        IF NOT fbSdoRead.bBusy THEN //nur starten wenn nicht bussy
			fbSdoRead(sNetId:= sNetId,nSlaveAddr :=nSlaveAddr, nIndex:=nIndex,
				nSubIndex :=nSubIndex, pDstBuf:= ADR(SlaveName), cbBufLen:=SIZEOF(SlaveName), bExecute:=TRUE);
			
            state := eStates.EXECUTING;
			ADSLOGSTR(
        	msgCtrlMask := ADSLOG_MSGTYPE_HINT, 
        	msgFmtStr   := 'set state executing %s','');
        END_IF
		//TODO TIMEOUT

    eStates.EXECUTING:
	
		fbSdoRead(); //Bussy flag update

		IF fbSdoRead.bBusy THEN
			// Warten auf Abschluss der Operation
		ELSE
            IF NOT fbSdoRead.bError THEN
                bReadSlaveNameSuccessful := TRUE;
											ADSLOGSTR(
        	msgCtrlMask := ADSLOG_MSGTYPE_HINT, 
        	msgFmtStr   := 'beendet ohne fehler %s','');
            ELSE
                bReadSlaveNameSuccessful := FALSE;
				bError := fbSdoRead.bError;
				nErrId := fbSdoRead.nErrId;
							ADSLOGSTR(
        	msgCtrlMask := ADSLOG_MSGTYPE_HINT, 
        	msgFmtStr   := 'beendet mit fehler %s','');
            END_IF
			
			IF SlaveName = RevSlaveName THEN
				bNameIsEqual := TRUE;
			ELSE
				bNameIsEqual := FALSE;
			END_IF
			
			bReadSlaveNameOccurred := TRUE; // Signalisieren, dass eine Änderung stattgefunden hat
			
            state := eStates.DONE;
        END_IF

    eStates.DONE:
	
	bExecute := FALSE;
    //waiting for reset ...  no automatic reset    
    //state := eStates.INIT;

ELSE
	state := eStates.INIT;
	
		
END_CASE;

{attribute 'TcRpcEnable'}
METHOD CheckName : BOOL
VAR_INPUT
		RevSlaveName : STRING;
END_VAR
bExecute := TRUE;
THIS^.RevSlaveName := RevSlaveName;
END_METHOD

METHOD FB_init : BOOL
VAR_INPUT
    bInitRetains : BOOL; // if TRUE, the retain variables are initialized (warm start / cold start)
    bInCopyCode  : BOOL; // if TRUE, the instance afterwards gets moved into the copy code (online change)
	sNetId           : T_AmsNetId;
END_VAR
THIS^.sNetId := sNetId;
END_METHOD

{attribute 'TcRpcEnable'}
METHOD Reset : BOOL
VAR_INPUT
END_VAR
state := eStates.INIT;
END_METHOD

END_FUNCTION_BLOCK
